FUNCTION_BLOCK FB_ISKRA_T6
// FB Utilisée uniquement pour motherfucking ISKRA de mes couilles.... 
// 
VAR_INPUT

	WORD_WEAK		: WORD;				// Strong Word. Word to consider if size equals 1.
	WORD_STRONG		: WORD;
END_VAR
VAR_OUTPUT
	VAR_OUT			: REAL;
END_VAR
VAR
	
	Filtre			: DWORD := 2#11111111000000000000000000000000;
	FullWord		: DWORD;
	ValExp			: SINT;
	ValCorps		: DINT;
	
END_VAR


FullWord := SHL(WORD_TO_DWORD(WORD_STRONG), 16) OR WORD_Weak;

ValExp := BYTE_TO_SINT(DWORD_TO_BYTE(SHR(FullWord, 24)));

ValCorps := -DWORD_TO_DINT(NOT (FullWord OR Filtre) + 1);


VAR_OUT :=  ValCorps*EXPT(10, ValExp);

END_FUNCTION_BLOCK

(* stored: Version 1.1.0.1, ProductVersion 3.1.4024.6
   POU FB_ISKRA_T6: Id {031d64bb-42bb-4f08-928f-da4340896024}, SpecialFunc None *)
